TYPE HMIRFIDControlInterface :
STRUCT
	ExecuteCommand	:	BOOL;
	SelectedCommand	:	WORD;
	SelectedMemoryIndex	:	WORD;
END_STRUCT
END_TYPE

(* stored: Version 1.1.0.1
   DUT HMIRFIDControlInterface: Id {552c278b-4581-4bf4-a1dc-5fd4902fa588} *)
